Staubli VAL3: lockAdvMove.pgx

program lockAdvMove(num x_nIndex)
begin
  //setMutex(bAdvMoves)
  bAdvMoveBusy[x_nIndex]=true
  //bAdvMoves=false
end
